INTERFACE I_Cylinder

PROPERTY Error : BOOL
GET
END_GET
END_PROPERTY

METHOD Extend
VAR_INPUT
END_VAR
END_METHOD

PROPERTY Extended : BOOL
GET
END_GET
END_PROPERTY

METHOD Retract
VAR_INPUT
END_VAR
END_METHOD

PROPERTY Retracted : BOOL
GET
END_GET
END_PROPERTY

END_INTERFACE

(* stored: Version 1.1.0.1, ProductVersion 3.1.4024.15
   Itf I_Cylinder: Id {5eef6192-44e5-0f9f-3fe7-0d8e658e50b6}
   Property Error: Id {a26df717-6531-4ed0-8404-a70bf4cf7959}
   Get Get: Id {672106fb-a426-4319-ab1f-83b1f2c9b639}
   Method Extend: Id {6199c781-0269-09a7-1ca0-96654d2c0840}
   Property Extended: Id {9168958e-d017-0813-27ac-c9aa4feccc2e}
   Get Get: Id {02c5faf0-ce44-0130-0631-7cd44984288e}
   Method Retract: Id {e7d61adf-37fc-023b-3604-04cdf6efdf9e}
   Property Retracted: Id {dde4e34a-b314-0277-079f-cf89835c0d08}
   Get Get: Id {4d086068-97be-0f17-0547-20f40cad0236} *)
